TEXTLIST TL_E_APP_VARIANT
  0 = 'INVALID'
  1 = 'VARIANT_OUTPUT_24'
  2 = 'VARIANT_OUTPUT_CLAMP'
   = ''
END_TEXTLIST

(* stored: Version 1.1.0.1
   TextList TL_E_APP_VARIANT: Id {c22ae4c5-0eed-4a37-bca8-ff113d61811f} *)
